// this script check the state functions and assigns the respective state value 

FUNCTION wr_GL_STATE : INT
VAR_INPUT
	TypeFunction : INT; // function
	State: INT;
END_VAR


//see folder state variables into GVLS folder for more details 
// -1 means that the robots just execute one specific state

//CASE TypeFunction OF
//	FUNCTION_PRG.TEST:
//	  	wr_GL_STATE:= -1;
//	FUNCTION_PRG.NORM:
//      	wr_GL_STATE:= State;
//	FUNCTION_PRG.MOVEMENTS:
//		wr_GL_STATE:= State;
//    FUNCTION_PRG.CK_COMUNICATIONS:
//		wr_GL_STATE:= -1;
//	FUNCTION_PRG.POWEROFF:
//		wr_GL_STATE:= State;
//END_CASE

END_FUNCTION

(* stored: Version 1.1.0.1, ProductVersion 3.1.4024.4
   POU wr_GL_STATE: Id {5c999248-76cb-4324-99a7-6c0d4b978838}, SpecialFunc None *)
